VAR_GLOBAL CONSTANT
	STRIP_LENGTH : UDINT := 12;
END_VAR

(* stored: Version 1.1.0.1
   GVL GVL: Id {a1b2c3d4-e5f6-7890-abcd-ef1234567890} *)
